// TwinCAT 3 PLC project PLC
// ProgramVersion: 3.1.4024.0
// libraries:
//   Tc2_Standard, * (Beckhoff Automation GmbH)
//   Tc2_System, * (Beckhoff Automation GmbH)
//   Tc2_Utilities, * (Beckhoff Automation GmbH)
//   Tc3_IotBase, * (Beckhoff Automation GmbH)
//   Tc3_Module, * (Beckhoff Automation GmbH)
//   Util, * (System)
// project tree:
//   Diagnostic/ GVL_Diagnostic.TcGVL (not stored), ST_Diagnostic.TcDUT (not stored)
//   FLM/Corking/ FB_CorkingRotation.TcPOU (not stored), E_FLM_CorkingStep.TcDUT (not stored), FB_FLM_CorkingStateMachine.TcPOU (not stored), ST_FLM_CorkingParams.TcDUT (not stored), ST_FLM_CorkingStatus.TcDUT (not stored)
//   FLM/Enums/ E_FLM_Step.TcDUT (not stored)
//   FLM/FBs/ FB_FLM_Diagnostic.TcPOU, FB_FLM_ReadCmd.TcPOU, FB_FLM_ReadCtrl.TcPOU, FB_FLM_ReadInputs.TcPOU (not stored), FB_FLM_ResetCmd.TcPOU (not stored), FB_FLM_WriteOutputs.TcPOU (not stored), FB_FLM_StateMachine.TcPOU
//   FLM/ FB_FLM_Main.TcPOU
//   FLM/Functions/ F_FLM_RawToLevel.TcPOU (not stored)
//   FLM/Structs/ ST_FLM_Cmd.TcDUT (not stored), ST_FLM_Ctrl.TcDUT (not stored), ST_FLM_In.TcDUT (not stored), ST_FLM_Motion.TcDUT (not stored), ST_FLM_Out.TcDUT, ST_FLM_Params.TcDUT (not stored), ST_FLM_RawIn.TcDUT, ST_FLM_RawOut.TcDUT, ST_FLM_Status.TcDUT, ST_FLM_StatusSaved.TcDUT (not stored)
//   / GlobalTextList.TcGTLO (not stored), IotTask.TcTTO, PlcTask.TcTTO, SimuTask.TcTTO, VisualizationManager.TcVMO (not stored)
//   GVLs/ GVL_IOT.TcGVL, GVL_PLC.TcGVL, GVL_SIMU.TcGVL
//   IOT/Enums/ E_IOT_DataType.TcDUT (not stored), E_IOT_Step.TcDUT (not stored), E_IOT_UpdateSpeed.TcDUT (not stored)
//   IOT/ FB_IOT.TcPOU, GVL_IOT_Constants.TcGVL (not stored)
//   IOT/Functions/ F_IOT_GetPayload.TcPOU, F_IOT_IsValueEqual.TcPOU
//   IOT/Structs/ ST_IOT_Data.TcDUT (not stored), ST_IOT_Params.TcDUT, ST_IOT_PeriodicPublishData.TcDUT (not stored), ST_IOT_OnChangePublishData.TcDUT (not stored)
//   IOT/Unions/ U_IOT_DataValue.TcDUT (not stored)
//   POUs/ IOT_MAIN.TcPOU, PLC_MAIN.TcPOU, SIMU_MAIN.TcPOU
//   Simulation/ FB_VisuSim.TcPOU
//   StateMachinePro/ E_Step.TcDUT (not stored), FB_StateMachinePro.TcPOU (not stored)
//   StateMachine/ FB_StateMachine.TcPOU (not stored)
//   VISUs/ Visu.TcVIS
// real-time tasks:
//   TASK IotTask: cycle T#1ms, priority 21, ADS port 350
//   TASK PlcTask: cycle T#1ms, priority 20, ADS port 351
//   TASK SimuTask: cycle T#10ms, priority 22, ADS port 352

CONFIGURATION PLC
    RESOURCE PLC ON TwinCAT3
        TASK IotTask(INTERVAL := T#1ms, PRIORITY := 21);
        TASK PlcTask(INTERVAL := T#1ms, PRIORITY := 20);
        TASK SimuTask(INTERVAL := T#10ms, PRIORITY := 22);
        PROGRAM IOT_MAIN WITH IotTask : IOT_MAIN;
        PROGRAM PLC_MAIN WITH PlcTask : PLC_MAIN;
        PROGRAM SIMU_MAIN WITH SimuTask : SIMU_MAIN;
    END_RESOURCE
END_CONFIGURATION

// ---- FLM/Structs/ST_FLM_Out.TcDUT
(* -----------------------------------------------------------------------------
| This sample has been supplied by Beckhoff As-Is and is intended only as an   |
| example implementation. Functionality is not guaranteed.                     |
----------------------------------------------------------------------------- *)

TYPE ST_FLM_Out :
STRUCT
	bFixedYellow : BOOL;		// luce gialla fissa
	bBlinkingYellow : BOOL;		// luce gialla lampeggiante
	bFixedGreen : BOOL;			// luce verde fissa
	bBlinkingGreen : BOOL;		// luce verde lampeggiante
	bHorn : BOOL;				// sirena di segnalazione
	
	bConveyor : BOOL;			// nastro trasportatore
	
	bWater : BOOL;				// riempimento acqua
	bMint : BOOL;				// riempimento menta	
	
	bCorkingVertical : BOOL;	// inserimento del tappo - movimento verticale
	bCorkingRotation : BOOL;	// inserimento del tappo - rotazione
END_STRUCT
END_TYPE

// ---- FLM/Structs/ST_FLM_RawIn.TcDUT
(* -----------------------------------------------------------------------------
| This sample has been supplied by Beckhoff As-Is and is intended only as an   |
| example implementation. Functionality is not guaranteed.                     |
----------------------------------------------------------------------------- *)

TYPE ST_FLM_RawIn :
STRUCT
	(* digital *)
	bEmergency AT %I*: BOOL;						// emergenza (NC)
	bStartButton  AT %I* : BOOL;					// pulsante di start (NO)
	bStopButton : BOOL;						// pulsante di stop (NC)
	bAckButton : BOOL;						// pulsante di riconoscimento allarmi (NO)
	bBottle : BOOL;							// fotocellula presenza bottiglia (NO)
	bCorkingRotationLimitSwitch : BOOL;		// finecorsa rotazione tappatura (NO)
	(* analog *)
	nWaterLevel : INT;						// livello acqua
	nMintLevel : INT;						// livello menta
END_STRUCT
END_TYPE

// ---- FLM/Structs/ST_FLM_RawOut.TcDUT
(* -----------------------------------------------------------------------------
| This sample has been supplied by Beckhoff As-Is and is intended only as an   |
| example implementation. Functionality is not guaranteed.                     |
----------------------------------------------------------------------------- *)

TYPE ST_FLM_RawOut :
STRUCT
	bConveyor  AT %Q* : BOOL;			// nastro trasportatore
	bWater  AT %Q* : BOOL;				// riempimento acqua
	bMint : BOOL;				// riempimento menta	
	bYellow : BOOL;				// luce gialla
	bGreen : BOOL;				// luce verde
	bHorn : BOOL;				// sirena di segnalazione
	bCorkingVertical : BOOL;	// inserimento del tappo - movimento verticale
	bCorkingRotation : BOOL;	// inserimento del tappo - rotazione
END_STRUCT
END_TYPE

// ---- FLM/Structs/ST_FLM_Status.TcDUT
(* -----------------------------------------------------------------------------
| This sample has been supplied by Beckhoff As-Is and is intended only as an   |
| example implementation. Functionality is not guaranteed.                     |
----------------------------------------------------------------------------- *)

TYPE ST_FLM_Status :
STRUCT
	
	stSaved : ST_FLM_StatusSaved;		// Valori ritenuti - utili p.e. per statistiche
	bCritical : BOOL;					// la macchina ha almento una condizione critica attiva
	bError : BOOL;						// la macchina ha almento una condizione di errore attiva	
	bWarning : BOOL;					// la macchina ha almeno una segnalazione attiva	
	bInfo : BOOL;						// la macchina ha almeno una informazione attiva			
	bVerbose : BOOL;					// la macchina ha almeno un messaggio attiva
	
	bFailure : BOOL;					// la macchina è in avaria (critica + error)	
	eStep : E_FLM_Step;					// passo della macchina a stati
	strStep : STRING;					// passo come stringa
	tStepTime : TIME;					// tempo di permanenza nel passo
	eErrorStep : E_FLM_Step;			// passo in cui si è generato l'errore
	nErrorID : DINT;					// codice di errore
	
	stCorking : ST_FLM_CorkingStatus;	// struttura di stato del dispositivo di tappatura
	
END_STRUCT
END_TYPE

// ---- IOT/Structs/ST_IOT_Params.TcDUT
(* -----------------------------------------------------------------------------
| This sample has been supplied by Beckhoff As-Is and is intended only as an   |
| example implementation. Functionality is not guaranteed.                     |
----------------------------------------------------------------------------- *)

// Questa struttura cointiene i parametri necessari al funzionamento della
// FB_IOT. 

TYPE ST_IOT_Params :
STRUCT
	// i parametri per instaurare la connessione con il broker 
	sHostName : STRING := 'test.mosquitto.org';
	nHostPort : UINT := 1883; 
	// certificati necessari per l'autenticazione. Si possono usare anche
	// user e password. vd: https://infosys.beckhoff.com/content/1033/tf6701_tc3_iot_communication_mqtt/3391835403.html?id=6531035858226877065
	
	stMqttTls : ST_IotMqttTls := ();
		
	// topic generale all'interno del quale ci saranno i subtopic nei quali
	// verranno pubblicati i dati
	// il pragma {attribute 'TcEncoding':='UTF-8'} va sempre usato per le 
	// stringhe quando si opera con MQTT
	{attribute 'TcEncoding':='UTF-8'}
	sTopicPrefix : STRING := 'FillerMachine';
	
	// subtopic da sottoscrivere per leggere i comandi  
	{attribute 'TcEncoding':='UTF-8'}
	sCmdSubscribedTopic : STRING := '/cmd';
	
	// numero massimo di messaggi da leggere per ciclo dai topic sottoscritti 
	nDequeueMessagesPerCycle : UINT := 3;
END_STRUCT
END_TYPE

// ---- GVLs/GVL_IOT.TcGVL
(* -----------------------------------------------------------------------------
| This sample has been supplied by Beckhoff As-Is and is intended only as an   |
| example implementation. Functionality is not guaranteed.                     |
----------------------------------------------------------------------------- *)

{attribute 'qualified_only'}
VAR_GLOBAL PERSISTENT
	stIotParams : ST_IOT_Params;		// Parametri per la comunicazione MQTT
	stFlmCmd : ST_FLM_Cmd;				// comandi di FLM
END_VAR

// ---- GVLs/GVL_PLC.TcGVL
(* -----------------------------------------------------------------------------
| This sample has been supplied by Beckhoff As-Is and is intended only as an   |
| example implementation. Functionality is not guaranteed.                     |
----------------------------------------------------------------------------- *)

{attribute 'qualified_only'}
VAR_GLOBAL PERSISTENT	
	stFlmParams : ST_FLM_Params;
	stFlmStatusSaved : ST_FLM_StatusSaved;	
END_VAR

VAR_GLOBAL
	bTaskRunning : BOOL;

	stFlmDiagnostic	: ST_Diagnostic;

	stFlmIn : ST_FLM_In;
	stFlmRawIn : ST_FLM_RawIn;
	stFlmOut : ST_FLM_Out;
	stFlmRawOut : ST_FLM_RawOut;
	stFlmCtrl : ST_FLM_Ctrl;	
	stFlmStatus : ST_FLM_Status;
	stFlmMotion	: ST_FLM_Motion;

END_VAR

// ---- GVLs/GVL_SIMU.TcGVL
{attribute 'qualified_only'}
VAR_GLOBAL
	bTaskRunning : BOOL;
END_VAR

// ---- POUs/IOT_MAIN.TcPOU
(* -----------------------------------------------------------------------------
| This sample has been supplied by Beckhoff As-Is and is intended only as an   |
| example implementation. Functionality is not guaranteed.                     |
----------------------------------------------------------------------------- *)

PROGRAM IOT_MAIN
VAR
	bInitialized : BOOL;
	bConnect : BOOL;		// richiesta TRUE -> connetti FALSE -> disconnetti
	
	// array per i dati da pubblicare e loro dimensione 
	aPeriodicPublish : ARRAY[0..GVL_IOT_Constants.cIOTMAXDATA - 1] OF ST_IOT_PeriodicPublishData;
	aOnChangePublish : ARRAY[0..GVL_IOT_Constants.cIOTMAXDATA - 1] OF ST_IOT_OnChangePublishData;		
	nPeriodicPublishSize : UDINT;	
	nOnChangePublishSize : UDINT;	
	
	fbIot : FB_IOT;
	nInitCycles : UDINT;
END_VAR

(* -----------------------------------------------------------------------------
| This sample has been supplied by Beckhoff As-Is and is intended only as an   |
| example implementation. Functionality is not guaranteed.                     |
----------------------------------------------------------------------------- *)

IF NOT bInitialized THEN
	IF nInitCycles = 0 THEN	
		ACT_InitPeriodic();	
		ACT_InitOnChange();
	END_IF;
	nInitCycles := nInitCycles + 1;
	bConnect := TRUE;
	bInitialized := GVL_PLC.bTaskRunning;	
ELSE
	
	// Qui vengono letti ad ogni ciclo i valori da FLM che verranno pubblicati
	// nei topic corrispondenti
 
	aOnChangePublish[0].stData.uValue.n := TO_DINT(GVL_PLC.stFlmStatus.eStep);
	aOnChangePublish[1].stData.uValue.b := GVL_PLC.stFlmStatus.bFailure;
	aOnChangePublish[2].stData.uValue.b := GVL_PLC.stFlmStatus.bWarning;

	aPeriodicPublish[0].stData.uValue.b := GVL_PLC.stFlmOut.bCorkingVertical;
	aPeriodicPublish[1].stData.uValue.b := GVL_PLC.stFlmOut.bCorkingRotation;
	aPeriodicPublish[2].stData.uValue.f := TO_LREAL(GVL_PLC.stFlmIn.fWaterLevel);
	aPeriodicPublish[3].stData.uValue.f := TO_LREAL(GVL_PLC.stFlmIn.fMintLevel);
	
	fbIot(
		bEnable:= TRUE, 
		bConnect:= bConnect, 
		tAutoAckTime:= T#2M, 
		stParams:= GVL_IOT.stIotParams, 
		aPeriodicPublish := aPeriodicPublish,		
		aOnChangePublish := aOnChangePublish,
		nPeriodicPublishSize := nPeriodicPublishSize, 
		nOnChangePublishSize := nOnChangePublishSize
	);
	
	// I comandi letti nel subtopic corrispondente vengono qui scritti su
	// delle variabili globali in modo da poter essere letti dalla task PLC
	// e usati all'interno di FLM
	GVL_IOT.stFlmCmd.bStart := fbIot.bFlmStartCmd;
	GVL_IOT.stFlmCmd.bStop := fbIot.bFlmStopCmd;
	GVL_IOT.stFlmCmd.bAck := fbIot.bFlmAckCmd;
END_IF

ACTION ACT_InitOnChange:
(* -----------------------------------------------------------------------------
| This sample has been supplied by Beckhoff As-Is and is intended only as an   |
| example implementation. Functionality is not guaranteed.                     |
----------------------------------------------------------------------------- *)

// inizializzazione degli elementi dell'array che contiene i dati da scambiare
// al cambiamento

aOnChangePublish[0].stData.sSubtopic := '/Step';
aOnChangePublish[0].stData.eType := E_IOT_DataType.I32;

aOnChangePublish[1].stData.sSubtopic := '/Failure';
aOnChangePublish[1].stData.eType := E_IOT_DataType.Boolean;

aOnChangePublish[2].stData.sSubtopic := '/Warning';
aOnChangePublish[2].stData.eType := E_IOT_DataType.Boolean;

// dimensione effettiva dell'array
nOnChangePublishSize := 3;
END_ACTION

ACTION ACT_InitPeriodic:
(* -----------------------------------------------------------------------------
| This sample has been supplied by Beckhoff As-Is and is intended only as an   |
| example implementation. Functionality is not guaranteed.                     |
----------------------------------------------------------------------------- *)

// inizializzazione degli elementi dell'array che contiene i dati da scambiare
// ciclicamente.

aPeriodicPublish[0].eUpdateSpeed := E_IOT_UpdateSpeed.Fast;
aPeriodicPublish[0].stData.sSubtopic := '/CorkingVertical';
aPeriodicPublish[0].stData.eType := E_IOT_DataType.Boolean;

aPeriodicPublish[1].eUpdateSpeed := E_IOT_UpdateSpeed.Fast;
aPeriodicPublish[1].stData.sSubtopic := '/CorkingRotation';
aPeriodicPublish[1].stData.eType := E_IOT_DataType.Boolean;

aPeriodicPublish[2].eUpdateSpeed := E_IOT_UpdateSpeed.Slow;
aPeriodicPublish[2].stData.sSubtopic := '/WaterLevel';
aPeriodicPublish[2].stData.eType := E_IOT_DataType.F64;

aPeriodicPublish[3].eUpdateSpeed := E_IOT_UpdateSpeed.Slow;
aPeriodicPublish[3].stData.sSubtopic := '/MintLevel';
aPeriodicPublish[3].stData.eType := E_IOT_DataType.F64;

// dimensione effettiva dell'array
nPeriodicPublishSize := 4;
END_ACTION

END_PROGRAM

// ---- IOT/FB_IOT.TcPOU
(* -----------------------------------------------------------------------------
| This sample has been supplied by Beckhoff As-Is and is intended only as an   |
| example implementation. Functionality is not guaranteed.                     |
----------------------------------------------------------------------------- *)

FUNCTION_BLOCK FB_IOT

VAR_INPUT
	bEnable : BOOL;						// abilitazione della FB
	bConnect : BOOL;					// bit che richiede la connessione
	tAutoAckTime : TIME;				// tempo di auto riconoscimento degli errori
	stParams : ST_IOT_Params;			// paramteri 
	nPeriodicPublishSize : UDINT;		// dimensione dell'array che continene i dati da pubblicare a tempo
	nOnChangePublishSize : UDINT;		// dimensione dell'arra che contiene i dati da pubblicare al cambiamento
END_VAR

VAR_IN_OUT
	aPeriodicPublish : ARRAY[0..GVL_IOT_Constants.cIOTMAXDATA - 1] OF ST_IOT_PeriodicPublishData;	// array di dati da pubblicare a tempo
	aOnChangePublish : ARRAY[0..GVL_IOT_Constants.cIOTMAXDATA - 1] OF ST_IOT_OnChangePublishData;	// array di dati da pubblicare al cambiamento
END_VAR

VAR_OUTPUT
	eStep :  E_IOT_Step;		// passo della macchina a stati
	tStepTime : TIME;			// tempo nel passo
	eErrStep : E_IOT_Step;		// passo in cui si è generato l'errore
	nErrId : DINT;				// id dell'errore
	bFlmStartCmd : BOOL;		// comando di start per FLM
	bFlmStopCmd : BOOL;			// comando di stop per FLM
	bFlmAckCmd : BOOL;			// comando di Ack per FLM
END_VAR

VAR
	bInitialized :  BOOL;
	eNewstep :  E_IOT_Step;
	bEntryact :  BOOL;
	fbTonStep :  TON;	
	bForceOnChangePublish : BOOL;	// forza la pubblicazione dei dati al cambiamento (acnhe se non sono cambiati)
	bMqttConnect : BOOL;			// bit di connessione MQTT
	udi : UDINT;
	fbMqttClient : FB_IotMqttClient;			// client MQTT	
	fbMessageQueue : FB_IotMqttMessageQueue;	// coda dei messaggi in ingresso	
	fbMessage : FB_IotMqttMessage;				// messaggio
	sPayload : STRING(255);
	bIsEqual : BOOL;	
	fbBlinkFast : BLINK;						// blink per la pubblicazione dati veloci
	fbBlinkSlow : BLINK;						// blinck pubblicazione dati lenti
	fbRtFast : R_TRIG;							// trigger pubblicazione dati veloci
	fbRtSlow : R_TRIG;							// trigger pubblicazione dati lenti
	bCmdTopicSubscribed : BOOL;	
	nDequeueCnt : UINT := 0;					// contatore di scodamento
	{attribute 'TcEncoding':='UTF-8'}
	sTopicRcv : STRING(255);					
	{attribute 'TcEncoding':='UTF-8'}
	sPayloadRcv : STRING(255);	
	{attribute 'TcEncoding':='UTF-8'}
	sAppo: STRING(255);	
	nFlmCmd : UINT := 0;
	fbTpFlmStartCmd : TP;						// impulso comando start FLM
	fbTpFlmStopCmd : TP;						// impulso comando start FLM
	fbTpFlmAckCmd : TP;							// impulso comando start FLM
END_VAR

(* -----------------------------------------------------------------------------
| This sample has been supplied by Beckhoff As-Is and is intended only as an   |
| example implementation. Functionality is not guaranteed.                     |
----------------------------------------------------------------------------- *)

// Questa macchina a stati serve per gestire la connessione verso il broker,
// la pubblicazione dei dati e la lettura dei messaggi nei topic sottoscritti.
// Tutto si basa su una FB di tipo FB_IotMqttClient
// https://infosys.beckhoff.com/content/1033/tf6701_tc3_iot_communication_mqtt/3391835403.html?id=6531035858226877065
// FB_IotMqttClient utilizza il paradigma della programmazione ad oggetti
// e in sostanza è una classe. Senza addentrarsi in una spiegazione della
// programmazione ad oggetti basti dire che una istanza di questa FB è un
// oggetto sul quale possono essere chiamati dei metodi. I metodi sono delle 
// funzioni proprie dell'oggetto specifico (l'istanza di FB_IotMqttClient) che
// hanno visibilità sulle variabili locali dell'oggetto. Ciascun metodo ha 
// la sua uscita, i suoi ingressi e le sue proprie variabili locali (temporanee)
// ma può anche operare sulle variabili locali dell'oggetto (l'istanza) che non 
// sono temporanee ma mantengono il valore tra una chiamata e l'altra. In 
// questo modo metodi diversi possono condividere delle aree di memoria che 
// altro non è che quella definita nelle variabili locali dell'oggetto.


IF NOT bInitialized THEN
	eNewstep := E_IOT_Step.NoStep;
	eStep := E_IOT_Step.Stop;
	bEntryact := FALSE;
	bInitialized := TRUE;		
ELSE	
	(* disabilitata o avaria *)	
	IF NOT bEnable THEN
		eNewstep := E_IOT_Step.NeOrError;
	END_IF
	
	IF eNewstep <> E_IOT_Step.NoStep THEN
		eStep := eNewstep;
		eNewstep := E_IOT_Step.NoStep;
		bEntryact := FALSE;
	END_IF;

	(* filtri *)	
	
	(* fronti *)	
	
	// questi blink e trigger servono a creare due bit (i trigger fast e slow)
	// che sono a TRUE solo per un ciclo ogni, rispettivamente, 100ms e 1s
	fbBlinkFast(ENABLE:= TRUE, TIMELOW:= T#50MS , TIMEHIGH:= T#50MS);	
	fbBlinkSlow(ENABLE:= TRUE, TIMELOW:= T#5S , TIMEHIGH:= T#5S);
	fbRtFast(CLK := fbBlinkFast.OUT);	
	fbRtSlow(CLK := fbBlinkSlow.OUT);
	
	(* richieste *)
	
	CASE eStep OF
		
		(* not Enabled or Error *)
		E_IOT_Step.NeOrError :
			(* entry action *)
			IF NOT bEntryact THEN
				bEntryact := TRUE;
			END_IF;

			(* body *)
			bMqttConnect := FALSE;
			bCmdTopicSubscribed := FALSE;
					
			(* transition *)
			IF bEnable THEN	
				IF tStepTime > tAutoAckTime THEN 		
					// qui si fa sostanzialmente un autoreset invece che lasciare 
					// tutto bloccato fino ad un intervento umano. Questa scelta si 
					// può fare per le funzionalitàù di comunicazione ma va sempre 
					// ben ponderata. Qui per esempio si valuta che è preferibile 
					// tentare di riconnettersi e che perdere informazioni sulle 
					// casuse di errore non è molto importante.
					eNewstep := E_IOT_Step.Reset;
				END_IF
			END_IF

			(* exitact *)
			IF eNewstep <> E_IOT_Step.NoStep THEN
				nErrId := 0;
				eErrStep := E_IOT_Step.NoStep;
			END_IF;

		(* Reset *)
		E_IOT_Step.Reset :
			(* entry action *)
			IF NOT bEntryact THEN				
				bEntryact := TRUE;
			END_IF;

			(* body *)
			bMqttConnect := FALSE;
					
			(* transition *)
			IF bEnable THEN				
				eNewstep := E_IOT_Step.Stop;				
			END_IF

			(* exitact *)
			IF eNewstep <> E_IOT_Step.NoStep THEN
				;
			END_IF;		
			
		(* Stop *)
		E_IOT_Step.Stop:
			(* entry action *)
			IF NOT bEntryact THEN
				bEntryact := TRUE;
			END_IF;

			(* body *)
			bMqttConnect := FALSE;			
							
			(* transition *)
			IF fbMqttClient.bError THEN
				eNewstep := E_IOT_Step.NeOrError;
			ELSE			
				IF bConnect THEN
					eNewstep := E_IOT_Step.Configure;
				END_IF
			END_IF
			
			(* exitact *)
			IF eNewstep <> E_IOT_Step.NoStep THEN
				IF eNewstep = E_IOT_Step.NeOrError THEN
					eErrStep := eStep;
					nErrID := fbMqttClient.hrErrorCode;				
				END_IF
			END_IF;
			
		(* Configure *)
		E_IOT_Step.Configure:
			(* entry action *)
			IF NOT bEntryact THEN
				bEntryact := TRUE;
			END_IF;

			(* body *)			
			fbMqttClient.sHostName:= stParams.sHostName;
			fbMqttClient.nHostPort:= stParams.nHostPort;
			//fbMqttClient.sClientId:= 'FLM'; 
			fbMqttClient.sTopicPrefix:= stParams.sTopicPrefix; 			 
			fbMqttClient.stTLS:= stParams.stMqttTls;
			fbMqttClient.nKeepAlive := 30;			
			fbMqttClient.ipMessageQueue := fbMessageQueue;			// FB che gestisce la coda di messaggi			
			bMqttConnect := FALSE;
							
			(* transition *)
			IF fbMqttClient.bError THEN
				eNewstep := E_IOT_Step.NeOrError;
			ELSE			
				eNewstep := E_IOT_Step.Connect;
			END_IF
			
			(* exitact *)
			IF eNewstep <> E_IOT_Step.NoStep THEN
				IF eNewstep = E_IOT_Step.NeOrError THEN
					eErrStep := eStep;
					nErrID := fbMqttClient.hrErrorCode;
				END_IF
			END_IF;
			
		(* Connect *)
		E_IOT_Step.Connect:
			(* entry action *)
			IF NOT bEntryact THEN
				bEntryact := TRUE;
			END_IF;

			(* body *)
			bMqttConnect := TRUE;
		
			(* transition *)
			IF fbMqttClient.bError THEN
				eNewstep := E_IOT_Step.NeOrError;
			ELSE
				IF bConnect THEN
					IF fbMqttClient.bConnected THEN
						eNewstep := E_IOT_Step.Subscribe;
					END_IF
				ELSE
					eNewstep := E_IOT_Step.Disconnect;	
				END_IF
			END_IF;
			
			(* exitact *)
			IF eNewstep <> E_IOT_Step.NoStep THEN
				IF eNewstep = E_IOT_Step.NeOrError THEN
					eErrStep := eStep;
					nErrID := fbMqttClient.hrErrorCode;
				END_IF
			END_IF;
			
		(* Subscribe *)
		E_IOT_Step.Subscribe:
			(* entry action *)
			IF NOT bEntryact THEN
				bCmdTopicSubscribed := FALSE;
				bEntryact := TRUE;
			END_IF;

			(* body *)
			bMqttConnect := TRUE;
			
			// questo metodo realizza la sottoscrizione al topic indicato
			// con la qualità del servizio indicata. 
			// (per QoS vedi: https://mosquitto.org/man/mqtt-7.html)
			bCmdTopicSubscribed := fbMqttClient.Subscribe(
				sTopic:=stParams.sCmdSubscribedTopic, 
				eQoS:=TcIotMqttQos.AtMostOnceDelivery			// qualità del servizo
			);
		
			(* transition *)
			IF fbMqttClient.bError OR NOT bCmdTopicSubscribed THEN
				eNewstep := E_IOT_Step.NeOrError;
			ELSE
				IF fbMqttClient.bConnected THEN
					eNewstep := E_IOT_Step.Online;
				END_IF
			END_IF;
			
			(* exitact *)
			IF eNewstep <> E_IOT_Step.NoStep THEN
				IF eNewstep = E_IOT_Step.NeOrError THEN
					eErrStep := eStep;
					nErrID := fbMqttClient.hrErrorCode;
				END_IF
			END_IF;
			
		(* Online *)
		E_IOT_Step.Online:
			(* entry action *)
			IF NOT bEntryact THEN	
				bForceOnChangePublish := TRUE;		
				bEntryact := TRUE;
			END_IF;

			(* body *)
			bMqttConnect := TRUE;
			ACT_PublishPeriodic();		// pubblicazione dati periodici
			ACT_PublishOnChange();		// pubblicazione dati al cambiamento
			ACT_DequeueMessages();		// lettura dei messaggi nei topic sottoscritti
		
			(* transition *)
			IF fbMqttClient.bError THEN
				eNewstep := E_IOT_Step.NeOrError;
			ELSE
				IF NOT bConnect THEN
					eNewstep := E_IOT_Step.Disconnect;
				END_IF
			END_IF;
			
			(* exitact *)
			IF eNewstep <> E_IOT_Step.NoStep THEN				
				IF eNewstep = E_IOT_Step.NeOrError THEN
					eErrStep := eStep;
					nErrID := fbMqttClient.hrErrorCode;
				END_IF
			END_IF;
			
		(* Unsubscribe *)
		E_IOT_Step.Unsubscribe:
			(* entry action *)
			IF NOT bEntryact THEN
				bCmdTopicSubscribed := FALSE;
				bEntryact := TRUE;
			END_IF;

			(* body *)
			bMqttConnect := TRUE;
			bCmdTopicSubscribed := NOT fbMqttClient.Unsubscribe(
				sTopic:=stParams.sCmdSubscribedTopic,				
			);
		
			(* transition *)
			IF fbMqttClient.bError OR NOT bCmdTopicSubscribed THEN
				eNewstep := E_IOT_Step.NeOrError;
			ELSE
				IF NOT bCmdTopicSubscribed THEN
					eNewstep := E_IOT_Step.Disconnect;
				END_IF
			END_IF;
			
			(* exitact *)
			IF eNewstep <> E_IOT_Step.NoStep THEN
				IF eNewstep = E_IOT_Step.NeOrError THEN
					eErrStep := eStep;
					nErrID := fbMqttClient.hrErrorCode;
				END_IF
			END_IF;
			
		(* Disconnect *)
		E_IOT_Step.Disconnect:
			(* entry action *)
			IF NOT bEntryact THEN
				bEntryact := TRUE;
			END_IF;

			(* body *)
			bMqttConnect := FALSE;
		
			(* transition *)
			IF fbMqttClient.bError THEN
				eNewstep := E_IOT_Step.NeOrError;
			ELSE
				IF NOT fbMqttClient.bConnected THEN
					eNewstep := E_IOT_Step.Stop;
				END_IF
			END_IF;
			
			(* exitact *)
			IF eNewstep <> E_IOT_Step.NoStep THEN
				IF eNewstep = E_IOT_Step.NeOrError THEN
					eErrStep := eStep;
					nErrID := fbMqttClient.hrErrorCode;
				END_IF
			END_IF;			
		ELSE
			eNewstep := E_IOT_Step.NeOrError;
			eErrStep := E_IOT_Step.Unknown;
			nErrId := -9;			
	END_CASE;
	
	(* tempo di permanenza nello step *)
	fbTonStep(IN := (eNewstep = E_IOT_Step.NoStep), PT := T#500H);
	tStepTime := fbTonStep.ET;
	
	(* FBs *)
	// questo metodo Execute va richiamato ad ogni ciclo. Si occupa di
	// instaurare e mantenere la connessione fino a quando l'ingresso 
	// passato è a TRUE	
	fbMqttClient.Execute(bMqttConnect);
	
	(* uscite *)
	fbTpFlmStartCmd(IN:= nFlmCmd = 1, PT:= T#200MS);
	fbTpFlmStopCmd(IN:= nFlmCmd = 2, PT:= T#200MS);
	fbTpFlmAckCmd(IN:= nFlmCmd = 3, PT:= T#200MS);
	bFlmStartCmd := fbTpFlmStartCmd.Q;
	bFlmStopCmd := fbTpFlmStopCmd.Q;
	bFlmAckCmd := fbTpFlmAckCmd.Q;

	
END_IF;

ACTION ACT_DequeueMessages:
(* -----------------------------------------------------------------------------
| This sample has been supplied by Beckhoff As-Is and is intended only as an   |
| example implementation. Functionality is not guaranteed.                     |
----------------------------------------------------------------------------- *)

// Questa action si occupa di verificare se ci sono messaggi nei subtopic 
// sottoscritti ed eventualmente di leggerli e decodificarli. 
// fbMessageQueue era stata precedentemente passata ad fbMqttClient in questo
// modo la coda può essere gestita dall'interno di fbMqttClient e anche 
// all'esterno.
// A sua volta fbMessage, che è una FB che serve a gestire il singolo messaggio
// viene passata a fbMessageQueue in modo che il messaggio sia gestibile sia 
// dall'interno di fbMessageQueue che dall'esterno.
// Se presente il messaggio viene scodato con fbMessageQueue.Dequeue poi
// si vanno a leggere il Topic e il payload con fbMessage.GetTopic  e
// fbMessage.GetPayload. Successivamente si estrapola dal topic completo
// solo la parte di subtopic che ci interessa per verifcare che corrisponda 
// al subtopic che abbiamo impostato nei parametri e solo a questo punto, 
// in base al valore del payload si prendono le azioni corrispondenti impostando
// la variabile nFlm a tre valori codificati (NB qui sarebbe stata una 
// buona idea usare una enumerazione... pazienza)

nFlmCmd := 0;
FOR nDequeueCnt := 0 TO stParams.nDequeueMessagesPerCycle - 1 DO
	IF fbMessageQueue.nQueuedMessages > 0 THEN
		IF fbMessageQueue.Dequeue(fbMessage:=fbMessage) THEN
			fbMessage.GetTopic(
					pTopic:=ADR(sTopicRcv), 
					nTopicSize:=SIZEOF(sTopicRcv)
			);
			fbMessage.GetPayload(
				pPayload:=ADR(sPayloadRcv), 
				nPayloadSize:=SIZEOF(sPayloadRcv),
				bSetNullTermination:=TRUE
			);
			
			 FindAndDelete(
				pSrcString:= ADR(sTopicRcv), 
				pDeleteString:= ADR(stParams.sTopicPrefix), 
				pDstString:= ADR(sAppo), 
				nDstSize:= SIZEOF(sAppo)
			);
			
			IF sAppo = stParams.sCmdSubscribedTopic THEN
				IF sPayloadRcv = 'start' THEN
					nFlmCmd := 1;
				ELSIF sPayloadRcv = 'stop' THEN
					nFlmCmd := 2;
				ELSIF sPayloadRcv = 'ack' THEN
					nFlmCmd := 3;
				END_IF
			END_IF
		END_IF
	END_IF	
END_FOR
END_ACTION

ACTION ACT_PublishOnChange:
(* -----------------------------------------------------------------------------
| This sample has been supplied by Beckhoff As-Is and is intended only as an   |
| example implementation. Functionality is not guaranteed.                     |
----------------------------------------------------------------------------- *)

// Questa Action si occupa della pubblicazione dei dati al cambiamento. Si cicla 
// tra gli elementi dell'array verificando che il dato sia cambiato per mezzo 
// di F_IOT_IsValueEqual. Se il dato è cambiato oppure la pubblicazione è 
// forzata tramite bForceOnChangePublish viene calcolato il payload con 
// F_IOT_GetPayload che converte il valore del dato in una stringa
// e lo si pubblica sul topic con il metodo Public di fbMqttClient.
// L'ingresso eQos indica la qualità richiesta per questa pubblicazione: in
// questo caso si desidera che la pubblicazione avvenga una e una sola volta, 
// senza duplicazioni. L'ingresso bRetain a TRUE fa in modo che il broker
// mantenga questa pubblicazione a disposizione per i client che si potrebbero 
// collegare in un secondo momento. Questa cosa ha senso visto che i dati 
// pubblicati al cambiamento potrebbero non cambiare per un tempo lungo e si 
// lascerebbe il client senza indicazioni per molto.

FOR udi := 0 TO nOnChangePublishSize - 1 DO
	bIsEqual :=  F_IOT_IsValueEqual(aOnChangePublish[udi].stData.eType, 
									aOnChangePublish[udi].stData.uValue, 
									aOnChangePublish[udi].uOldValue);
	IF bForceOnChangePublish OR NOT bIsEqual THEN
														
		F_IOT_GetPayload(aOnChangePublish[udi].stData, ADR(sPayload), SIZEOF(sPayload));
		fbMqttClient.Publish(
					sTopic:= aOnChangePublish[udi].stData.sSubtopic, 
					pPayload:= ADR(sPayload), 
					nPayloadSize:= LEN2(ADR(sPayload)), 
					eQoS:= TcIotMqttQos.AtMostOnceDelivery, 
					bRetain:= TRUE,								 // !
					bQueue:= FALSE
		);
		aOnChangePublish[udi].uOldValue := aOnChangePublish[udi].stData.uValue;
	END_IF	
END_FOR

bForceOnChangePublish := FALSE;
END_ACTION

ACTION ACT_PublishPeriodic:
(* -----------------------------------------------------------------------------
| This sample has been supplied by Beckhoff As-Is and is intended only as an   |
| example implementation. Functionality is not guaranteed.                     |
----------------------------------------------------------------------------- *)

// Questa Action si occupa della pubblicazione dei dati periodici. Si cicla 
// tra gli elementi dell'array distinguendo tra i dati con pubblicazione veloce
// e quelli a pubblicazione lenta e verificando la presenza del trigger
// corrispondente. Se le condizioni sono soddisfate si calcola il payload con 
// F_IOT_GetPayload che converte il valore del dato in una stringa e  lo si 
// pubblica sul topic con il metodo Public di fbMqttClient.
// L'ingresso eQos indica la qualità richiesta per questa pubblicazione: in
// questo caso si desidera che la pubblicazione avvenga una e una sola volta, 
// senza duplicazioni. L'ingresso bRetain a FALSE fa in modo che il broker non
// mantenga questa pubblicazione a disposizione per i client che si potrebbero 
// collegare in un secondo momento. 

FOR udi := 0 TO nPeriodicPublishSize - 1 DO
	IF fbRtFast.Q AND aPeriodicPublish[udi].eUpdateSpeed = E_IOT_UpdateSpeed.Fast THEN	
		F_IOT_GetPayload(aPeriodicPublish[udi].stData, ADR(sPayload), SIZEOF(sPayload));
		fbMqttClient.Publish(
				sTopic:= aPeriodicPublish[udi].stData.sSubtopic, 
				pPayload:= ADR(sPayload), 
				nPayloadSize:= LEN2(ADR(sPayload)), 
				eQoS:= TcIotMqttQos.AtMostOnceDelivery, 
				bRetain:= FALSE,
				bQueue:= FALSE
		);
	END_IF;	
	
	IF fbRtSlow.Q AND aPeriodicPublish[udi].eUpdateSpeed = E_IOT_UpdateSpeed.Slow THEN	
		F_IOT_GetPayload(aPeriodicPublish[udi].stData, ADR(sPayload), SIZEOF(sPayload));
		fbMqttClient.Publish(
				sTopic:= aPeriodicPublish[udi].stData.sSubtopic, 
				pPayload:= ADR(sPayload), 
				nPayloadSize:= LEN2(ADR(sPayload)), 
				eQoS:= TcIotMqttQos.AtMostOnceDelivery, 
				bRetain:= FALSE,
				bQueue:= FALSE
		);
	END_IF;
END_FOR
END_ACTION

END_FUNCTION_BLOCK

// ---- IOT/Functions/F_IOT_IsValueEqual.TcPOU
(* -----------------------------------------------------------------------------
| This sample has been supplied by Beckhoff As-Is and is intended only as an   |
| example implementation. Functionality is not guaranteed.                     |
----------------------------------------------------------------------------- *)

// Questa funzione confronta il valore attuale del dato con il suo valore 
// precedente.  Anche qui si vede l'utilità dell'unione: se non si fosse 
// utilizzata l'unione sarebbero state necessarie tre  funzioni molto simili 
// che differivano solamente per il tipo di dato in ingresso.

FUNCTION F_IOT_IsValueEqual : BOOL
VAR_INPUT
	eType : E_IOT_DataType;
	uVal1 : U_IOT_DataValue;
	uVal2 : U_IOT_DataValue;	
END_VAR
VAR
END_VAR


IF eType = E_IOT_DataType.Boolean THEN
	F_IOT_IsValueEqual := uVal1.b = uVal2.b;
ELSIF eType = E_IOT_DataType.F64 THEN
	F_IOT_IsValueEqual := uVal1.f = uVal2.f;
ELSIF eType = E_IOT_DataType.I32 THEN
F_IOT_IsValueEqual := uVal1.n = uVal2.n;
ELSE
	F_IOT_IsValueEqual := FALSE;	
END_IF

END_FUNCTION

// ---- IOT/Functions/F_IOT_GetPayload.TcPOU
(* -----------------------------------------------------------------------------
| This sample has been supplied by Beckhoff As-Is and is intended only as an   |
| example implementation. Functionality is not guaranteed.                     |
----------------------------------------------------------------------------- *)

// Questa funzione calcola il Payload del dato. Il Payload altro non è che la
// rappresentazione del valore come stringa. Qui si vede l'utilità dell'unione
// se non si fosse utilizziata l'unione sarebbero state necessarie tre 
// funzioni molto simili che differivano solamente per il tipo di dato in 
// ingresso.


FUNCTION F_IOT_GetPayload : BOOL
VAR_INPUT
	stDataValue : ST_IOT_Data;
	pPayload : POINTER TO STRING;
	nSize : UDINT;
END_VAR
VAR
	bRes : BOOL;
	sAppo1 : STRING(255);	
END_VAR

(* -----------------------------------------------------------------------------
| This sample has been supplied by Beckhoff As-Is and is intended only as an   |
| example implementation. Functionality is not guaranteed.                     |
----------------------------------------------------------------------------- *)

IF stDataValue.eType = E_IOT_DataType.Boolean THEN 
	sAppo1 := TO_STRING(stDataValue.uValue.b);
ELSIF stDataValue.eType = E_IOT_DataType.F64 THEN
	sAppo1 := TO_STRING(stDataValue.uValue.f);
ELSE
	sAppo1 := TO_STRING(stDataValue.uValue.n);
END_IF
	
F_IOT_GetPayload := STRNCPY(pPayload, ADR(sAppo1), nSize);

END_FUNCTION

// ---- POUs/PLC_MAIN.TcPOU
(* -----------------------------------------------------------------------------
| This sample has been supplied by Beckhoff As-Is and is intended only as an   |
| example implementation. Functionality is not guaranteed.                     |
----------------------------------------------------------------------------- *)

PROGRAM PLC_MAIN
VAR
	bInitialized : BOOL;
	
	fbGetCurTaskIndex : GETCURTASKINDEX;		
	tTaskCycleTime : UDINT;					// tempo di ciclo della task in microsecondi
	tTaskExecTime : UDINT;					// tempo di esecuzione della task in microsecondi
	tTaskMaxExecTime : UDINT;				// tempo massimo di esecuzione della task in microsecondi

	fbFlm : FB_FLM_Main;
	
	
	// fbTest : FB_FLM_CorkingStateMachine;
END_VAR

(* -----------------------------------------------------------------------------
| This sample has been supplied by Beckhoff As-Is and is intended only as an   |
| example implementation. Functionality is not guaranteed.                     |
----------------------------------------------------------------------------- *)

IF NOT bInitialized THEN
	
	// Get the Cycle Time of the task to which this PRG is assigned (it will then be shared with the State Machine)
	fbGetCurTaskIndex();
	tTaskCycleTime := _TaskInfo[fbGetCurTaskIndex.index].CycleTime / 10;	// CycleTime is expressed in multiples of 100ns
	bInitialized := GVL_SIMU.bTaskRunning;
	
ELSE
	
	(* task time *)
	tTaskExecTime := _TaskInfo[fbGetCurTaskIndex.index].LastExecTime / 10;		// ExecTime is expressed in multiples of 100ns
	IF tTaskExecTime > tTaskMaxExecTime THEN
			tTaskMaxExecTime := tTaskExecTime;
	END_IF;	
	
	(* machine *)
		
	fbFlm(
		bEnable:= TRUE, 
		tTaskCycleTime:= tTaskCycleTime, 
		nId:= 0, 
		bHwError:= FALSE,	
		stRawIn := GVL_PLC.stFlmRawIn,
		stIn := GVL_PLC.stFlmIn,
		stRawOut := GVL_PLC.stFlmRawOut,
		stOut := GVL_PLC.stFlmOut,
		stCtrl := GVL_PLC.stFlmCtrl,		
		stParams := GVL_PLC.stFlmParams,
		stDiagnostic := GVL_PLC.stFlmDiagnostic,
		stStatus := GVL_PLC.stFlmStatus,
		stStatusSaved := GVL_PLC.stFlmStatusSaved,
		stMotion := GVL_PLC.stFlmMotion,
		stIotCmd := GVL_IOT.stFlmCmd	 
	);
		
	
		
	(* 
	fbTest(
		bEnable:= TRUE, 
		bAck:= GVL_PLC.stFlmIn.bAckButton, 
		bStart:= GVL_PLC.stFlmIn.bStartButton, 
		bStop:= GVL_PLC.stFlmIn.bStopButton, 
		bRotationLimitSwitch:= GVL_PLC.stFlmIn.bCorkingRotationLimitSwitch, 
		stParams:= GVL_PLC.stFlmParams.stCorking, 
	);
	*)
	
	GVL_PLC.bTaskRunning := TRUE;
END_IF

END_PROGRAM

// ---- FLM/FB_FLM_Main.TcPOU
(* -----------------------------------------------------------------------------
| This sample has been supplied by Beckhoff As-Is and is intended only as an   |
| example implementation. Functionality is not guaranteed.                     |
----------------------------------------------------------------------------- *)

FUNCTION_BLOCK FB_FLM_Main

VAR_INPUT
	bEnable			: BOOL;
	tTaskCycleTime	: UDINT;
	nId				: USINT;	
	bHwError		: BOOL;	
END_VAR

VAR_OUTPUT

END_VAR
	
VAR_IN_OUT
	stRawIn : ST_FLM_RawIn;
	stIn : ST_FLM_In;	
	stRawOut : ST_FLM_RawOut;
	stOut : ST_FLM_Out;
	stCtrl : ST_FLM_Ctrl;	
	stParams : ST_FLM_Params;
	stDiagnostic : ST_Diagnostic;
	stStatus : ST_FLM_Status;
	stStatusSaved : ST_FLM_StatusSaved;
	stMotion : ST_FLM_Motion;
	stIotCmd : ST_FLM_Cmd;

END_VAR

VAR
	bInitialized : BOOL;
	stCmd : ST_FLM_Cmd;
	errno : INT;
	(* fbReadPar : fbMachineReadPars; *)
	fbReadCmd : FB_FLM_ReadCmd;
	fbResetCmd : FB_FLM_ResetCmd;
	fbReadCtrl : FB_FLM_ReadCtrl;
	fbReadIn : FB_FLM_ReadInputs;
	fbDiagnostic : FB_FLM_Diagnostic;
	fbStateMachine : FB_FLM_StateMachine;
	fbCorkingStateMachine : FB_FLM_CorkingStateMachine;
	
	fbWriteOut : FB_FLM_WriteOutputs;
	
END_VAR

(* -----------------------------------------------------------------------------
| This sample has been supplied by Beckhoff As-Is and is intended only as an   |
| example implementation. Functionality is not guaranteed.                     |
----------------------------------------------------------------------------- *)

IF NOT bInitialized THEN
	stStatus.stSaved := stStatusSaved;
	bInitialized := TRUE;		
ELSE

	(* 01 - Leggi ingressi, controlli, parametri e comandi  *)	
	fbReadIn(
		stParams := stParams,		
		stRawIn := stRawIn
	);				
	
	stIn := fbReadIn.stIn;
	fbReadCtrl(
		nId := nId,	
		bEnable := bEnable,
		stIn := stIn,	
				
	);
	stCtrl := fbReadCtrl.stCtrl;
		
	fbReadCmd(
		stIn := stIn, 
		stIotCmd := stIotCmd
	);
	stCmd := fbReadCmd.stCmd;	

	(* 03 - Gestione eventi *)	
	fbDiagnostic(
		stIn := stIn,
		stOut := stOut,
		stCtrl := stCtrl,
		stParams := stParams,
		bHwError := bHwError, 
		bAck := stCmd.bAck, 
		stStatus := stStatus, 
		stMotion := stMotion,
		stDiagnostic := stDiagnostic, 
	);
	stStatus.bCritical := fbDiagnostic.bCritical;
	stStatus.bError := fbDiagnostic.bError;
	stStatus.bWarning := fbDiagnostic.bWarning;
	stStatus.bInfo := fbDiagnostic.bInfo;
	stStatus.bVerbose := fbDiagnostic.bVerbose;
	stStatus.bFailure := fbDiagnostic.bFailure;
	
	stOut.bBlinkingYellow := fbDiagnostic.bBlinking;
	stOut.bFixedYellow := fbDiagnostic.bFixed;
	stOut.bHorn := fbDiagnostic.bHorn;

	(* 04 - Macchina a stati principale: *)		
	fbStateMachine(
		stIn := stIn,
		stCtrl := stCtrl,
		stCmd := stCmd,
		stParams := stParams,
		stStatus := stStatus,		
		bBottle := stIn.bBottle,
	);	
	stStatus.eStep := fbStateMachine.eStep;
	stStatus.strStep := TO_STRING(stStatus.eStep);
	stStatus.tStepTime := fbStateMachine.tStepTime;
	stStatus.eErrorStep := fbStateMachine.eErRstep; 
	stStatus.nErrorID := fbStateMachine.nErrId;
	
	stOut.bConveyor := fbStateMachine.bConveyor;
	stOut.bWater := fbStateMachine.bWater;
	stOut.bMint := fbStateMachine.bMint;
	stOut.bBlinkingGreen := fbStateMachine.bBlinkingGreen;
	stOut.bFixedGreen := fbStateMachine.bFixedGreen;
	
	(* 05 - Macchine a stati secondarie *)
	fbCorkingStateMachine(
		bEnable:= stCtrl.bEnable AND stCtrl.bEmergency AND NOT stStatus.bFailure,
		bAck:= stCmd.bAck, 
		bStart:= fbStateMachine.bCorkingStart, 
		bStop:= FALSE, // stCmd.bStop, 
		bRotationLimitSwitch:= stIn.bCorkingRotationLimitSwitch, 
		stParams:= stParams.stCorking,		 
	);
	stStatus.stCorking.eStep := fbCorkingStateMachine.eStep;
	stStatus.stCorking.tStepTime := fbCorkingStateMachine.tStepTime;
	stStatus.stCorking.eErrorStep := fbCorkingStateMachine.eErrStep;
	stStatus.stCorking.nErrorID	:= fbCorkingStateMachine.nErrID; 
	
	stOut.bCorkingRotation := fbCorkingStateMachine.bRotation;
	stOut.bCorkingVertical := fbCorkingStateMachine.bVertical;
	
	(* 06 - Scrivi uscite e informazioni *)	
	fbWriteOut(		
		stOut		:= stOut,
		stParams	:= stParams,		
		stRawOut	:= stRawOut
	);
	
	// stStatus.stSaved.nCounter := stStatus.stSaved.nCounter +1;	   
	
	stStatusSaved := stStatus.stSaved;		// aggiorna struttura con i dati salvati

	(* 07 - fine - altre operazioni*)
		
	// fbResetCmd();

END_IF;

END_FUNCTION_BLOCK

// ---- FLM/FBs/FB_FLM_ReadCmd.TcPOU
(* -----------------------------------------------------------------------------
| This sample has been supplied by Beckhoff As-Is and is intended only as an   |
| example implementation. Functionality is not guaranteed.                     |
----------------------------------------------------------------------------- *)

FUNCTION_BLOCK FB_FLM_ReadCmd

VAR_INPUT
	stIn : ST_FLM_In;
	stIotCmd : ST_FLM_Cmd;
END_VAR

VAR_OUTPUT
	stCmd : ST_FLM_Cmd;
END_VAR

VAR_IN_OUT
	
END_VAR

VAR
	fbRtStart	: R_TRIG;
	fbRtStop	: R_TRIG;
	fbTpAck		: TP;	
END_VAR
VAR CONSTANT
	
END_VAR

(* -----------------------------------------------------------------------------
| This sample has been supplied by Beckhoff As-Is and is intended only as an   |
| example implementation. Functionality is not guaranteed.                     |
----------------------------------------------------------------------------- *)

fbRtStart(CLK := stIn.bStartButton OR stIotCmd.bStart);
fbRtStop(CLK := stIn.bStopButton OR stIotCmd.bStop);
fbTpAck(IN:= stIn.bAckButton OR stIotCmd.bAck, PT:= T#200MS);


stCmd.bAck		:= fbTpAck.Q;
stCmd.bStop		:= fbRtStop.Q;
stCmd.bStart	:= fbRtStart.Q;

END_FUNCTION_BLOCK

// ---- FLM/FBs/FB_FLM_ReadCtrl.TcPOU
(* -----------------------------------------------------------------------------
| This sample has been supplied by Beckhoff As-Is and is intended only as an   |
| example implementation. Functionality is not guaranteed.                     |
----------------------------------------------------------------------------- *)

FUNCTION_BLOCK FB_FLM_ReadCtrl

VAR_INPUT
	nId:	INT;
	bEnable : BOOL;
	//stIn : ST_FLM_In;
END_VAR

VAR_IN_OUT
	stIn : ST_FLM_In;
END_VAR

VAR_OUTPUT
	stCtrl : ST_FLM_Ctrl;
END_VAR

VAR
	fbTonStartup: TON;
END_VAR

(* -----------------------------------------------------------------------------
| This sample has been supplied by Beckhoff As-Is and is intended only as an   |
| example implementation. Functionality is not guaranteed.                     |
----------------------------------------------------------------------------- *)

fbTonStartup(IN := TRUE, PT := T#3S);
stCtrl.bEmergency := stIn.bEmergency;
stCtrl.bEnable := fbTonStartup.Q AND bEnable;

END_FUNCTION_BLOCK

// ---- FLM/FBs/FB_FLM_Diagnostic.TcPOU
(* -----------------------------------------------------------------------------
| This sample has been supplied by Beckhoff As-Is and is intended only as an   |
| example implementation. Functionality is not guaranteed.                     |
----------------------------------------------------------------------------- *)

FUNCTION_BLOCK FB_FLM_Diagnostic
VAR_INPUT
	stIn : ST_FLM_In;
	stOut : ST_FLM_Out;
	stParams : ST_FLM_Params;
	stCtrl : ST_FLM_Ctrl;
	bHwError : BOOL;
	bAck : BOOL;
	stStatus : ST_FLM_Status;
END_VAR

VAR_IN_OUT
	stMotion : ST_FLM_Motion;
	stDiagnostic : ST_Diagnostic;
END_VAR

VAR_OUTPUT	
	bCritical : BOOL;
	bError : BOOL;
	bWarning : BOOL;
	bInfo  : BOOL;
	bVerbose : BOOL;
	bFailure : BOOL;
	bBlinking : BOOL;
	bFixed : BOOL;
	bHorn : BOOL;
END_VAR

VAR	
	stInstantDiagnostic : ST_Diagnostic;	
	nUi : UDINT;

END_VAR

(* -----------------------------------------------------------------------------
| This sample has been supplied by Beckhoff As-Is and is intended only as an   |
| example implementation. Functionality is not guaranteed.                     |
----------------------------------------------------------------------------- *)

(* reSet condizioni istantantanee *)
FOR nUi := 0 TO GVL_Diagnostic.cMAXEVENTS -1 DO
	stInstantDiagnostic.aCritical[nUi]	:= 0;
	stInstantDiagnostic.aError[nUi]		:= 0;
	stInstantDiagnostic.aWarning[nUi]	:= 0;
	stInstantDiagnostic.aInfo[nUi]		:= 0;
	stInstantDiagnostic.aVerbose[nUi]	:= 0; 
END_FOR

(* filtri, etc *)

(* imposta condizioni istantanee *)
stInstantDiagnostic.aCritical[0] := bHwError;
stInstantDiagnostic.aCritical[1] := NOT stCtrl.bEmergency;

stInstantDiagnostic.aError[0] := stStatus.eErrorStep <> E_FLM_Step.NoStep;
stInstantDiagnostic.aError[1] := stStatus.stCorking.eErrorStep <> E_FLM_CorkingStep.NoStep;
stInstantDiagnostic.aError[2] := (stStatus.eStep > E_FLM_Step.Stop) AND (stIn.fWaterLevel < stParams.fWaterMaxLevel * 0.1);
stInstantDiagnostic.aError[3] := (stStatus.eStep > E_FLM_Step.Stop) AND (stIn.fMintLevel < stParams.fMintMaxLevel * 0.1);

stInstantDiagnostic.aWarning[0] := (stStatus.eStep > E_FLM_Step.Stop) AND (stIn.fWaterLevel < stParams.fWaterMaxLevel * 0.2);
stInstantDiagnostic.aWarning[1] := (stStatus.eStep > E_FLM_Step.Stop) AND (stIn.fMintLevel < stParams.fMintMaxLevel * 0.2);

(* reset condizioni ritenute *)
IF bAck THEN
	FOR nUi := 0 TO GVL_Diagnostic.cMAXEVENTS -1 DO
		stDiagnostic.aCritical[nUi] := 0;
		stDiagnostic.aError[nUi] := 0;
		stDiagnostic.aWarning[nUi] := 0;
		stDiagnostic.aInfo[nUi] := 0;
		stDiagnostic.aVerbose[nUi] := 0; 
	END_FOR
	bCritical := FALSE;
	bError := FALSE;
	bWarning := FALSE;
	bInfo := FALSE;
	bVerbose := FALSE;
	bBlinking := FALSE;
	bHorn := FALSE;
END_IF									

(* imposta condizioni ritenute *)									
FOR nUi := 0 TO GVL_Diagnostic.cMAXEVENTS -1 DO
	IF stInstantDiagnostic.aCritical[nUi] THEN
		stDiagnostic.aCritical[nUi] := TRUE;
		bCritical := TRUE;
	END_IF
	IF stInstantDiagnostic.aError[nUi] THEN
		stDiagnostic.aError[nUi] := TRUE;
		bError := TRUE;
	END_IF
	IF stInstantDiagnostic.aWarning[nUi] THEN
		stDiagnostic.aWarning[nUi] := TRUE;
		bWarning := TRUE;
	END_IF
	IF stInstantDiagnostic.aInfo[nUi] THEN
		stDiagnostic.aInfo[nUi] := TRUE;
		bInfo := TRUE;
	END_IF
	IF stInstantDiagnostic.aVerbose[nUi] THEN
		stDiagnostic.aVerbose[nUi] := TRUE;
		bVerbose := TRUE;
	END_IF
END_FOR

bFailure := bCritical OR bError;

bBlinking := bFailure;
bHorn := bFailure;
bFixed := bWarning;

END_FUNCTION_BLOCK

// ---- FLM/FBs/FB_FLM_StateMachine.TcPOU
(* -----------------------------------------------------------------------------
| This sample has been supplied by Beckhoff As-Is and is intended only as an   |
| example implementation. Functionality is not guaranteed.                     |
----------------------------------------------------------------------------- *)

FUNCTION_BLOCK FB_FLM_StateMachine
VAR_INPUT	
	stIn		: ST_FLM_In;
	stCtrl		: ST_FLM_Ctrl;
	stCmd		: ST_FLM_Cmd;
	stParams	: ST_FLM_Params;
	stStatus	: ST_FLM_Status;
		
	bBottle : BOOL;				// fotocellula FC1
END_VAR

VAR_OUTPUT
	eStep :  E_FLM_Step;
	tStepTime : TIME;
	eErrStep : E_FLM_Step;
	nErrId : DINT;
	
	bConveyor : BOOL;			// nastro trasportatore
	bWater : BOOL;				// riempimento acqua
	bMint : BOOL;				// riempimento menta	
	bCorkingStart : BOOL;		// start inserimento del tappo	
	bBlinkingGreen : BOOL;		// lampada verde lampeggiante
	bFixedGreen : BOOL;			// lampada verde lampeggiante
END_VAR

VAR_IN_OUT
	
END_VAR

VAR
	bInitialized :  BOOL;
	eNewstep :  E_FLM_Step;
	bEntryact :  BOOL;
	fbTonStep :  TON;	
	
	fbTonBottle : TON;
	fbRtBottle : R_TRIG;
		
	bStopRequest : BOOL;
	
	nFillingCycles : USINT;
END_VAR

(* -----------------------------------------------------------------------------
| This sample has been supplied by Beckhoff As-Is and is intended only as an   |
| example implementation. Functionality is not guaranteed.                     |
----------------------------------------------------------------------------- *)

IF NOT bInitialized THEN
	eNewstep := E_FLM_Step.NoStep;
	eStep := E_FLM_Step.Stop;
	bEntryact := FALSE;
	bInitialized := TRUE;		
ELSE	
	(* disabilitata o avaria *)	
	IF NOT stCtrl.bEnable OR NOT(stCtrl.bEmergency) OR stStatus.bFailure THEN
		eNewstep := E_FLM_Step.NeOrError;
	END_IF
	
	IF eNewstep <> E_FLM_Step.NoStep THEN
		eStep := eNewstep;
		eNewstep := E_FLM_Step.NoStep;
		bEntryact := FALSE;
	END_IF;

	(* filtri *)
	fbTonBottle(IN:= bBottle, PT:= T#500MS);		// filtro sensore presenza bottiglia
	
	(* fronti *)
	fbRtBottle(CLK:= fbTonBottle.Q);
	
	(* richieste *)
	IF stCmd.bStop THEN
		bStopRequest := TRUE;
	END_IF; 
	
	CASE eStep OF
		
		(* not Enabled or Error *)
		E_FLM_Step.NeOrError :
			(* entry action *)
			IF NOT bEntryact THEN
				bEntryact := TRUE;
			END_IF;

			(* body *)
			bConveyor := FALSE;
			bWater := FALSE;
			bMint := FALSE;
			bCorkingStart := FALSE;
			bBlinkingGreen := FALSE;
			bFixedGreen := FALSE;
			
			nFillingCycles := 0;
					
			(* transition *)
			IF stCtrl.bEnable THEN				
				IF stCmd.bAck THEN
					eNewstep := E_FLM_Step.Reset;
				END_IF
			END_IF

			(* exitact *)
			IF eNewstep <> E_FLM_Step.NoStep THEN
				nErrId := 0;
				eErrStep := E_FLM_Step.NoStep;
			END_IF;

		(* Reset *)
		E_FLM_Step.Reset :
			(* entry action *)
			IF NOT bEntryact THEN				
				bEntryact := TRUE;
			END_IF;

			(* body *)
			bConveyor := FALSE;
			bWater := FALSE;
			bMint := FALSE;
			bCorkingStart := FALSE;
			bBlinkingGreen := FALSE;
			bFixedGreen := FALSE;
			
			nFillingCycles := 0;
					
			(* transition *)
			IF stCtrl.bEnable THEN				
				IF NOT stStatus.bFailure AND stStatus.stCorking.eStep = E_FLM_CorkingStep.Stop THEN
					eNewstep := E_FLM_Step.Stop;
				END_IF
			END_IF

			(* exitact *)
			IF eNewstep <> E_FLM_Step.NoStep THEN
				;
			END_IF;		
			
		(* Stop *)
		E_FLM_Step.Stop:
			(* entry action *)
			IF NOT bEntryact THEN
				bStopRequest := FALSE;
				bEntryact := TRUE;
			END_IF;

			(* body *)
			bConveyor := FALSE;
			bWater := FALSE;
			bMint := FALSE;
			bCorkingStart := FALSE;
			bBlinkingGreen := FALSE;
			bFixedGreen := FALSE;
			
			nFillingCycles := 0;
				
			(* transition *)			
			IF NOT stCmd.bStop AND stCmd.bStart THEN
				eNewstep := E_FLM_Step.Feeding;
			END_IF
			
			(* exitact *)
			IF eNewstep <> E_FLM_Step.NoStep THEN
				;
			END_IF;
			
		(* Feeding *)
		E_FLM_Step.Feeding:
			(* entry action *)
			IF NOT bEntryact THEN
				bEntryact := TRUE;
			END_IF;

			(* body *)
			bConveyor := TRUE;
			bWater := FALSE;
			bMint := FALSE;
			bCorkingStart := FALSE;
			bBlinkingGreen := FALSE;
			bFixedGreen := TRUE;
			bBlinkingGreen := bStopRequest;
			bFixedGreen := TRUE;
		
			(* transition *)
			IF bStopRequest AND NOT bBottle THEN
				eNewstep := E_FLM_Step.Stopping;
			ELSE
				IF fbRtBottle.Q THEN
					eNewstep := E_FLM_Step.WaterFilling;
				END_IF
			END_IF
			
			(* exitact *)
			IF eNewstep <> E_FLM_Step.NoStep THEN
				;
			END_IF;
			
		(* Water Filling *)
		E_FLM_Step.WaterFilling:
			(* entry action *)
			IF NOT bEntryact THEN
				nFillingCycles := nFillingCycles + 1;
				bEntryact := TRUE;
			END_IF;

			(* body *)
			bConveyor := FALSE;
			bWater := TRUE;
			bMint := FALSE;
			bCorkingStart := FALSE;
			bBlinkingGreen := bStopRequest;
			bFixedGreen := TRUE;
		
			(* transition *)
			IF tStepTime >= stParams.tWaterFillingTime THEN
				eNewstep := E_FLM_Step.MintFilling;
			END_IF
			
			(* exitact *)
			IF eNewstep <> E_FLM_Step.NoStep THEN
				;
			END_IF;
			
		(* Mint Filling *)
		E_FLM_Step.MintFilling:
			(* entry action *)
			IF NOT bEntryact THEN
				bEntryact := TRUE;
			END_IF;

			(* body *)
			bConveyor := FALSE;
			bWater := FALSE;
			bMint := TRUE;
			bCorkingStart := FALSE;
			bBlinkingGreen := bStopRequest;
			bFixedGreen := TRUE;
		
			(* transition *)
			IF tStepTime >= stParams.tMintFillingTime THEN
				IF nFillingCycles >= stParams.nFillingCycles THEN
					eNewstep := E_FLM_Step.Corking;
				ELSE 
					eNewstep := E_FLM_Step.WaterFilling;
				END_IF
					
			END_IF
			
			(* exitact *)
			IF eNewstep <> E_FLM_Step.NoStep THEN
				IF eNewstep = E_FLM_Step.Corking THEN
					nFillingCycles := 0;
				END_IF
			END_IF;	

		(* Corking *)
		E_FLM_Step.Corking:
			(* entry action *)
			IF NOT bEntryact THEN
				bEntryact := TRUE;
			END_IF;

			(* body *)
			bConveyor := FALSE;
			bWater := FALSE;
			bMint := FALSE;
			bCorkingStart := TRUE;
			bBlinkingGreen := bStopRequest;
			bFixedGreen := TRUE;
		
			(* transition *)
			IF stStatus.stCorking.eStep = E_FLM_CorkingStep.Done THEN
				eNewstep := E_FLM_Step.Feeding;
			END_IF
			
			(* exitact *)
			IF eNewstep <> E_FLM_Step.NoStep THEN
				;
			END_IF;

		(* Stopping *)
		E_FLM_Step.Stopping:
			(* entry action *)
			IF NOT bEntryact THEN
				bEntryact := TRUE;
			END_IF;

			(* body *)
			bConveyor := tStepTime < T#500MS;
			bWater := tStepTime >= T#1000MS AND tStepTime <= T#1300MS;
			bMint := tStepTime >= T#1000MS AND tStepTime <= T#1300MS;
			bCorkingStart := FALSE;
			bBlinkingGreen := TRUE;
			bFixedGreen := FALSE;
		
			(* transition *)
			IF tStepTime >= T#4S THEN
				eNewstep := E_FLM_Step.Stop;
			END_IF; 
			
			(* exitact *)
			IF eNewstep <> E_FLM_Step.NoStep THEN
				;
			END_IF;		
		ELSE
			eNewstep := E_FLM_Step.NeOrError;
			eErrStep := E_FLM_Step.Unknown;
			nErrId := -9;			
	END_CASE;
	
	(* tempo di permanenza nello step *)
	fbTonStep(IN := (eNewstep = E_FLM_Step.NoStep), PT := T#500H);
	tStepTime := fbTonStep.ET;
	
END_IF;

END_FUNCTION_BLOCK

// ---- POUs/SIMU_MAIN.TcPOU
(* -----------------------------------------------------------------------------
| This sample has been supplied by Beckhoff As-Is and is intended only as an   |
| example implementation. Functionality is not guaranteed.                     |
----------------------------------------------------------------------------- *)

PROGRAM SIMU_MAIN
VAR
	bInitialized : BOOL;
	fbVisuSim : FB_VisuSim;
	bRefillMint : BOOL;
	bRefillWater : BOOL;
	bEmergencyButton : BOOL;
	fPos : REAL;
END_VAR

(* -----------------------------------------------------------------------------
| This sample has been supplied by Beckhoff As-Is and is intended only as an   |
| example implementation. Functionality is not guaranteed.                     |
----------------------------------------------------------------------------- *)

IF NOT bInitialized THEN
	bEmergencyButton := TRUE;	
	bInitialized := TRUE;
	
ELSE
	(* Visu and Simulation *)
	fbVisuSim(
		bConveyor := GVL_PLC.stFlmRawOut.bConveyor, 
		bWater := GVL_PLC.stFlmRawOut.bWater, 
		bMint := GVL_PLC.stFlmRawOut.bMint,
		bCorkingRotation := GVL_PLC.stFlmRawOut.bCorkingRotation, 
		bCokingVertical := GVL_PLC.stFlmRawOut.bCorkingVertical,
		bRefillWater := bRefillWater, 
		bRefillMint := bRefillMint,
		bEmergencyButton := bEmergencyButton,
	);
	fpos := fbVisuSim.fPos;
	GVL_PLC.stFlmRawIn.bEmergency := fbVisuSim.bEmergency;
	GVL_PLC.stFlmRawIn.bBottle := fbVisuSim.bBottle;
	GVL_PLC.stFlmRawIn.nWaterLevel := fbVisuSim.nWaterLevel;
	GVL_PLC.stFlmRawIn.nMintLevel := fbVisuSim.nMintLevel;
	GVL_PLC.stFlmRawIn.bCorkingRotationLimitSwitch := fbVisuSim.bCorkingRotationLimitSwitch; 
	GVL_SIMU.bTaskRunning := TRUE;
END_IF

END_PROGRAM

// ---- Simulation/FB_VisuSim.TcPOU
(* -----------------------------------------------------------------------------
| This sample has been supplied by Beckhoff As-Is and is intended only as an   |
| example implementation. Functionality is not guaranteed.                     |
----------------------------------------------------------------------------- *)

FUNCTION_BLOCK FB_VisuSim
VAR_INPUT
	bConveyor : BOOL;
	bWater : BOOL;
	bMint : BOOL;
	bCorkingRotation : BOOL;
	bCokingVertical : BOOL;
	bRefillWater : BOOL;
	bRefillMint : BOOL;
	bEmergencyButton : BOOL;
END_VAR
VAR_OUTPUT
	fPos : REAL;	
	bBottle : BOOL;
	nWaterLevel : INT;
	nMintLevel : INT;
	bCorkingRotationLimitSwitch : BOOL;
	bEmergency : BOOL;
END_VAR
VAR
	bInitialized : BOOL;	
	nCorkingRotationCnt : UINT;
	nCorkingRotationCntLowerLimit : UINT := 30;
	fbRefill : BLINK;
	fbRtRefill : R_TRIG;
END_VAR

(* -----------------------------------------------------------------------------
| This sample has been supplied by Beckhoff As-Is and is intended only as an   |
| example implementation. Functionality is not guaranteed.                     |
----------------------------------------------------------------------------- *)

IF NOT bInitialized THEN
	nWaterLevel := 32000;
	nMintLevel := 24000;
	bInitialized := TRUE;	
ELSE
	
	(* Simulazione pulsante di emergenza *)
	bEmergency := bEmergencyButton;	
	
	(* simulazione nastro trasportatore e sensore presenza bottiglia *)
	IF bConveyor THEN
		fPos := fPos + 0.1;
	END_IF
	
	IF fPos >= 120.0 THEN
		fPos := 0;
	END_IF
	
	bBottle := fPos >= 60.0 AND fPos <= 80.0;
	
	(* simulazione auto-approvvigionamento liquidi *) 
	fbRefill(ENABLE:= TRUE, TIMELOW:= T#15S, TIMEHIGH:= T#15S);
	fbRtRefill(CLK := fbRefill.OUT);
	IF fbRtRefill.Q THEN
		IF nWaterLevel < 11000 THEN
			bRefillWater := TRUE;
		END_IF
		IF nMintLevel < 9000 THEN
			bRefillMint := TRUE;
		END_IF
	END_IF
	
	(* simulazione livelli acqua e menta *)
	IF bWater THEN
		nWaterLevel := nWaterLevel - 11;
	END_IF
	
	IF nWaterLevel < 0 THEN
		nWaterLevel := 0;
	END_IF
	
	IF bRefillWater THEN
		nWaterLevel := nWaterLevel + 19567;
	END_IF
	
	IF bMint THEN
		nMintLevel := nMintLevel - 17;
	END_IF
	
	IF nMintLevel < 0 THEN
		nMintLevel := 0;
	END_IF
	
	IF bRefillMint THEN
		nMintLevel := nMintLevel + 20231;
	END_IF
	
	bRefillWater := FALSE;
	bRefillMint := FALSE;
	
	(* simulazione sensore tappatura *)
	IF bCokingVertical THEN
		IF bCorkingRotation THEN
			nCorkingRotationCnt := nCorkingRotationCnt + 1;
		END_IF
	ELSE
		nCorkingRotationCnt := 0;
	END_IF
	
	bCorkingRotationLimitSwitch := nCorkingRotationCnt > nCorkingRotationCntLowerLimit;
	
	
	
	
	
	
	
	
	
END_IF

END_FUNCTION_BLOCK

// ---- VISUs/Visu.TcVIS
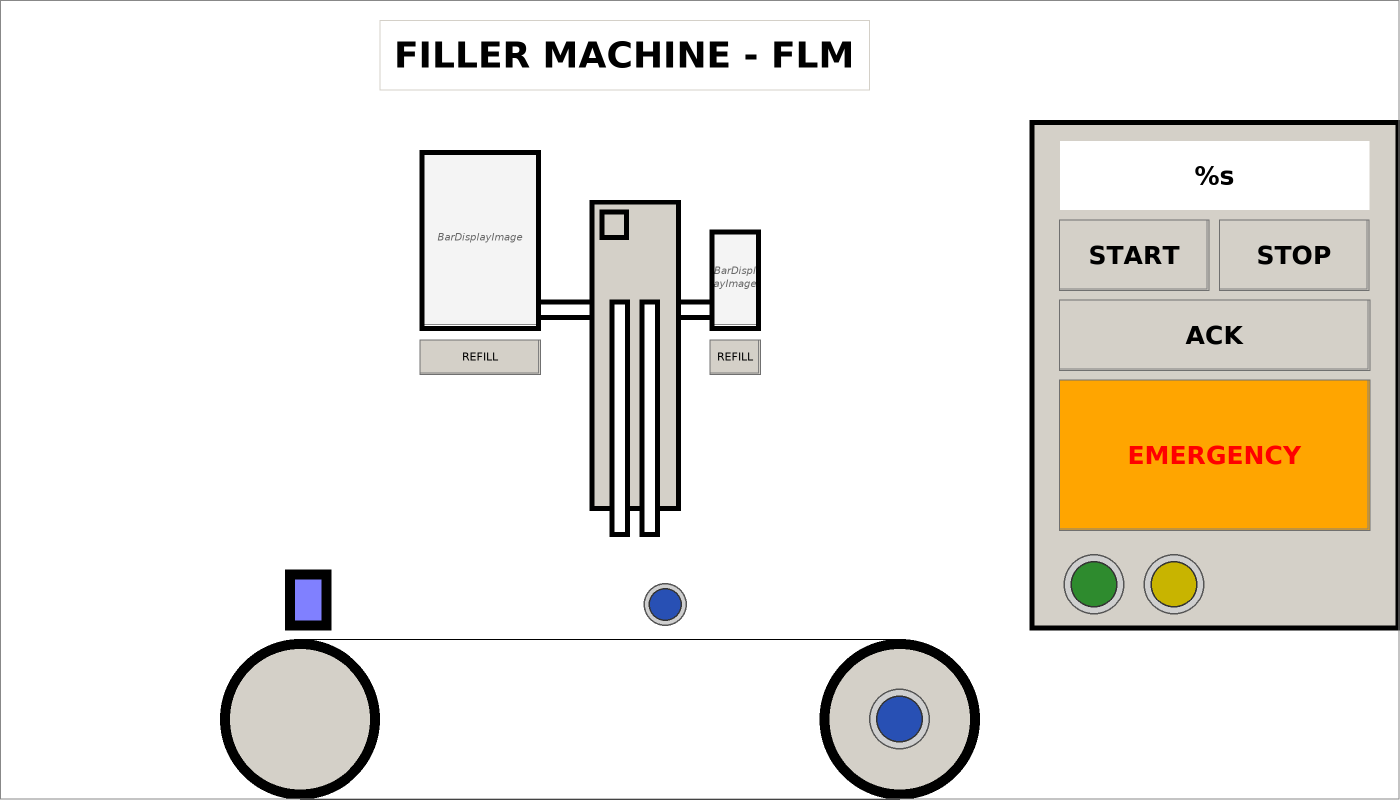
VISUALIZATION Visu  // 1401x801
    Rectangle (650,300 101x20), colour toggle: GVL_PLC.stFlmRawOut.bMint
    Rectangle (520,300 110x20), colour toggle: GVL_PLC.stFlmRawOut.bWater
    Rectangle (590,200 91x311), colour toggle: GVL_PLC.stFlmRawOut.bCorkingRotation
        p2738717112: (TO_REAL(GVL_PLC.stFlmRawOut.bCorkingVertical) * 50.0)
    Ellipse (220,640 160x160)
    Line (300,640) (900,640)
    Ellipse (820,640 160x160)
    Line (300,800) (900,800)
    Lamp1 (865,685 70x70), variable: GVL_PLC.stFlmRawOut.bConveyor, style: Lamp-Lamp1-Blue
    Rectangle (610,300 20x237), colour toggle: GVL_PLC.stFlmRawOut.bWater
    Rectangle (640,300 20x237), colour toggle: GVL_PLC.stFlmRawOut.bMint
    Lamp1 (640,580 51x50), variable: GVL_PLC.stFlmRawIn.bBottle, style: Lamp-Lamp1-Blue
    RoundedRectangle (285,570 46x61), invisible if: SIMU_MAIN.fPos > 100.0
        p3560616238: SIMU_MAIN.fPos * 5.0
    RoundedRectangle (1030,120 371x511)
    Button (1060,220 150x71), "START"
        tap GVL_PLC.stFlmRawIn.bStartButton
    Button (1220,220 150x71), "STOP"
        tap GVL_PLC.stFlmRawIn.bStopButton p1329445385=TRUE
    Textfield (1060,140 311x71), "%s", text variable: GVL_PLC.stFlmStatus.eStep
    Button (1060,300 311x71), "ACK"
        tap GVL_PLC.stFlmRawIn.bAckButton
    Button (1060,380 311x151), "EMERGENCY"
        toggle SIMU_MAIN.bEmergencyButton
    Group (710,230 51x101)
        BarDisplayImage (0,0 51x95), value: GVL_PLC.stFlmRawIn.nMintLevel, style: BarDisplayImage-Gray, scale format: %.1f, scale 0..32767
        Rectangle (0,0 51x101), colour toggle: GVL_PLC.stFlmRawOut.bCorkingRotation
    Group (420,150 121x181)
        BarDisplayImage (0,0 121x175), value: GVL_PLC.stFlmRawIn.nWaterLevel, style: BarDisplayImage-Gray, scale format: %.1f, scale 0..32767
        Rectangle (0,0 121x181), colour toggle: GVL_PLC.stFlmRawOut.bCorkingRotation
    RoundedRectangle (600,210 29x30), colour toggle: GVL_PLC.stFlmRawIn.bCorkingRotationLimitSwitch
        p2738717112: (TO_REAL(GVL_PLC.stFlmRawOut.bCorkingVertical) * 50.0)
    Button (420,340 121x35), "REFILL"
        tap SIMU_MAIN.bRefillWater
    Button (710,340 51x35), "REFILL"
        tap SIMU_MAIN.bRefillMint
    Lamp1 (1060,550 70x70), variable: GVL_PLC.stFlmRawOut.bGreen, style: Lamp-Lamp1-Green
    Lamp1 (1140,550 70x70), variable: GVL_PLC.stFlmRawOut.bYellow, style: Lamp-Lamp1-Yellow
    Textfield (380,20 490x70), "FILLER MACHINE - FLM"
END_VISUALIZATION
